Staubli VAL3: getTrajType.pgx

program getTrajType(string& x_sTrajType[])
  local num l_nPos
  local string l_sPath
begin
  // get the trajType
end
